// LS Electric XG5000 project: Timer2
// PLC NewPLC
// module base 0 slot 0: 입출력 모듈:XBC-DR20S (DC 24V 입력 12점, 릴레이 출력 8점)

PROGRAM NewProgram (task: 스캔 프로그램)

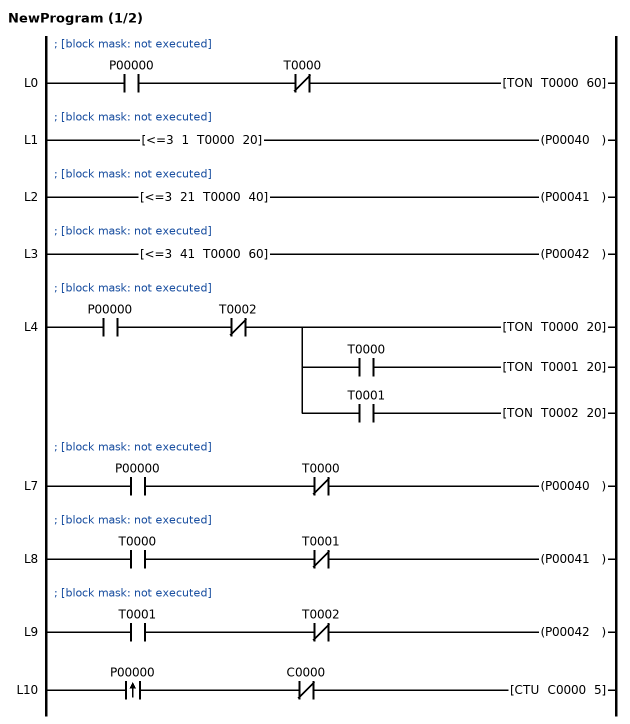
; L0 (block mask: not executed)
LOAD      P00000
AND NOT   T0000
TON       T0000 60
; L1 (block mask: not executed)
LOAD<=3   1 T0000 20
OUT       P00040
; L2 (block mask: not executed)
LOAD<=3   21 T0000 40
OUT       P00041
; L3 (block mask: not executed)
LOAD<=3   41 T0000 60
OUT       P00042
; L4 (block mask: not executed)
LOAD      P00000
AND NOT   T0002
TON       T0000 20
MPUSH
AND       T0000
TON       T0001 20
MPOP
AND       T0001
TON       T0002 20
; L7 (block mask: not executed)
LOAD      P00000
AND NOT   T0000
OUT       P00040
; L8 (block mask: not executed)
LOAD      T0000
AND NOT   T0001
OUT       P00041
; L9 (block mask: not executed)
LOAD      T0001
AND NOT   T0002
OUT       P00042
; L10
LOADP     P00000
AND NOT   C0000
CTU       C0000 5

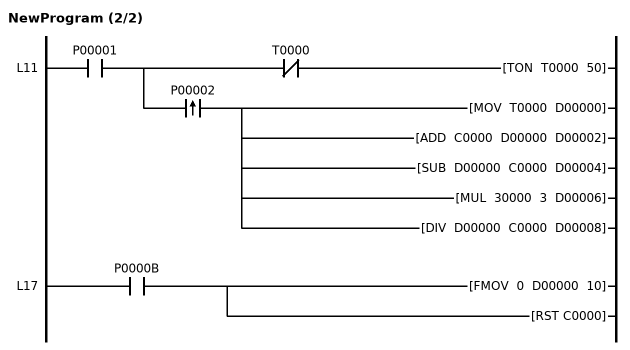
; L11
LOAD      P00001
MPUSH
AND NOT   T0000
TON       T0000 50
MPOP
ANDP      P00002
MOV       T0000 D00000
ADD       C0000 D00000 D00002
SUB       D00000 C0000 D00004
MUL       30000 3 D00006
DIV       D00000 C0000 D00008
; L17
LOAD      P0000B
FMOV      0 D00000 10
RST       C0000